FUNCTION_BLOCK FB_PU_les
VAR_INPUT
	Zustand_Lueftungsanlage	: ST_LA_Zustand;
END_VAR
VAR_OUTPUT
END_VAR
VAR
	IN_StatusModule			AT %I*: ARRAY [0..5] OF USINT;
	IN_Leistung				AT %I*: UDINT;		(* 0..100% *)

	IN_Leistung_elek		AT %I*: UDINT;	(* W *)
	IN_Leistung_therm		AT %I*: UDINT;	(* W *)
	IN_Energie_elek			AT %I*: UDINT;
	IN_Energie_therm		AT %I*: UDINT;
	IN_Volumenstrom			AT %I*: UDINT;
	IN_Volumen				AT %I*: UDINT;
	IN_Temp_intern			AT %I*: REAL;
	IN_Temp_extern			AT %I*: UDINT;
	IN_Temp_elek			AT %I*: UDINT;
	IN_Drehzahl				AT %I*: UDINT;	(* U/min *)
	IN_Frequenz_Motor		AT %I*: UDINT;	(* Hz *)
	IN_Zeit_Betrieb			AT %I*: UDINT;		(* h *)
	IN_Anzahl_Starts		AT %I*: UDINT;
	IN_Modul_Meld_Code1		AT %I*: USINT;
	IN_Modul_Meld_Code2		AT %I*: USINT;
	IN_Druckdifferenz		AT %I*: UDINT;


	IN_Temp_intern_GeniReply	AT %I*: ST_PU_Genibus;
	OUT_Temp_intern_GeniRequest	AT %Q*: ST_PU_Genibus;
	OUT_ControlModule	AT %Q*: ARRAY [0..4] OF USINT;
	{attribute 'OPC.UA.DA' := '1'}Zustand					: ST_PU_les_Zustand;	
	LeseDaten				: FB_PU_les_Input;
	StatusModul1			: DWORD;
	StatusModul2			: DWORD;
	ControlModul1			: DWORD;
	ControlModul2			: DWORD;
	Genibus					: FB_PU_les_Genibus;
END_VAR

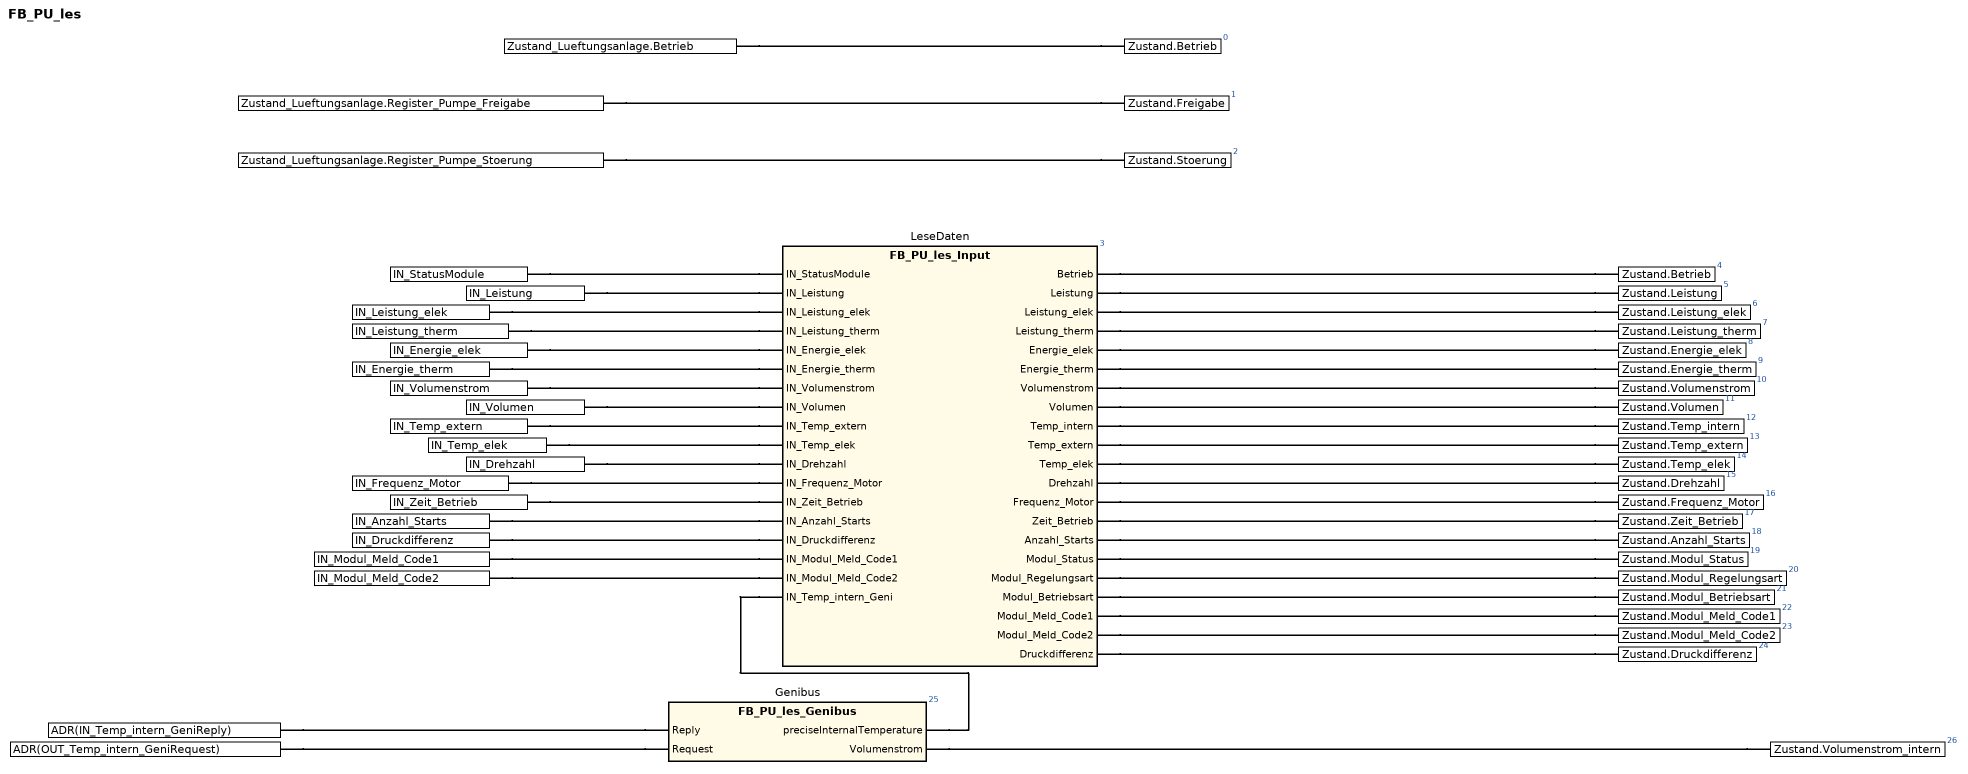
Zustand.Betrieb := Zustand_Lueftungsanlage.Betrieb;
Zustand.Freigabe := Zustand_Lueftungsanlage.Register_Pumpe_Freigabe;
Zustand.Stoerung := Zustand_Lueftungsanlage.Register_Pumpe_Stoerung;
LeseDaten(
    IN_StatusModule := IN_StatusModule,
    IN_Leistung := IN_Leistung,
    IN_Leistung_elek := IN_Leistung_elek,
    IN_Leistung_therm := IN_Leistung_therm,
    IN_Energie_elek := IN_Energie_elek,
    IN_Energie_therm := IN_Energie_therm,
    IN_Volumenstrom := IN_Volumenstrom,
    IN_Volumen := IN_Volumen,
    IN_Temp_extern := IN_Temp_extern,
    IN_Temp_elek := IN_Temp_elek,
    IN_Drehzahl := IN_Drehzahl,
    IN_Frequenz_Motor := IN_Frequenz_Motor,
    IN_Zeit_Betrieb := IN_Zeit_Betrieb,
    IN_Anzahl_Starts := IN_Anzahl_Starts,
    IN_Druckdifferenz := IN_Druckdifferenz,
    IN_Modul_Meld_Code1 := IN_Modul_Meld_Code1,
    IN_Modul_Meld_Code2 := IN_Modul_Meld_Code2,
    IN_Temp_intern_Geni := Genibus.preciseInternalTemperature); // FB_PU_les_Input
Zustand.Betrieb := LeseDaten.Betrieb;
Zustand.Leistung := LeseDaten.Leistung;
Zustand.Leistung_elek := LeseDaten.Leistung_elek;
Zustand.Leistung_therm := LeseDaten.Leistung_therm;
Zustand.Energie_elek := LeseDaten.Energie_elek;
Zustand.Energie_therm := LeseDaten.Energie_therm;
Zustand.Volumenstrom := LeseDaten.Volumenstrom;
Zustand.Volumen := LeseDaten.Volumen;
Zustand.Temp_intern := LeseDaten.Temp_intern;
Zustand.Temp_extern := LeseDaten.Temp_extern;
Zustand.Temp_elek := LeseDaten.Temp_elek;
Zustand.Drehzahl := LeseDaten.Drehzahl;
Zustand.Frequenz_Motor := LeseDaten.Frequenz_Motor;
Zustand.Zeit_Betrieb := LeseDaten.Zeit_Betrieb;
Zustand.Anzahl_Starts := LeseDaten.Anzahl_Starts;
Zustand.Modul_Status := LeseDaten.Modul_Status;
Zustand.Modul_Regelungsart := LeseDaten.Modul_Regelungsart;
Zustand.Modul_Betriebsart := LeseDaten.Modul_Betriebsart;
Zustand.Modul_Meld_Code1 := LeseDaten.Modul_Meld_Code1;
Zustand.Modul_Meld_Code2 := LeseDaten.Modul_Meld_Code2;
Zustand.Druckdifferenz := LeseDaten.Druckdifferenz;
Genibus(Reply := ADR(IN_Temp_intern_GeniReply), Request := ADR(OUT_Temp_intern_GeniRequest)); // FB_PU_les_Genibus
Zustand.Volumenstrom_intern := Genibus.Volumenstrom;

END_FUNCTION_BLOCK

(* stored: Version 1.1.0.1, ProductVersion 3.1.4024.9
   POU FB_PU_les: Id {5e3a26df-b1e7-41d6-9718-892ff736af86}, SpecialFunc None *)
